// LS Electric XG5000 project: 16-45-1
// PLC NewPLC
// module base 0 slot 0: 입출력 모듈:XBC-DR14E (DC 24V 입력 8점, 릴레이 출력 6점)

PROGRAM NewProgram (task: 스캔 프로그램)

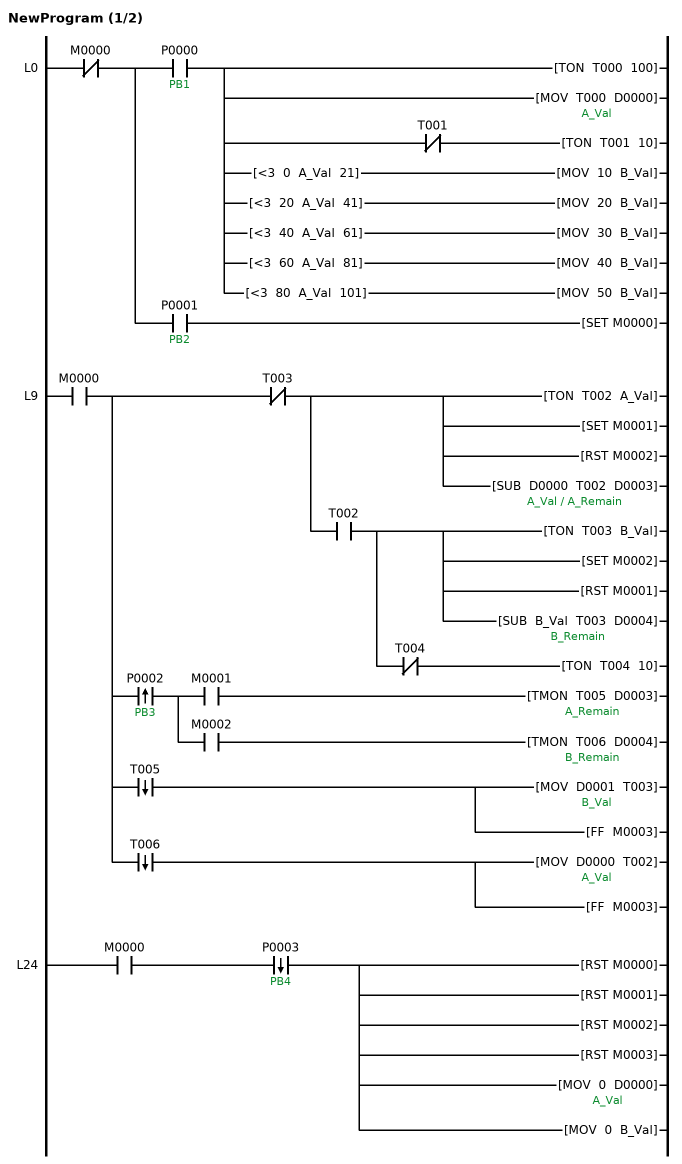
; L0
LOAD NOT  M0000
MPUSH
AND       P0000	// PB1
TON       T000 100
MOV       T000 D0000	// A_Val
MPUSH
AND NOT   T001
TON       T001 10
MLOAD
AND<3     0 A_Val 21
MOV       10 B_Val
MLOAD
AND<3     20 A_Val 41
MOV       20 B_Val
MLOAD
AND<3     40 A_Val 61
MOV       30 B_Val
MLOAD
AND<3     60 A_Val 81
MOV       40 B_Val
MPOP
AND<3     80 A_Val 101
MOV       50 B_Val
MPOP
AND       P0001	// PB2
SET       M0000
; L9
LOAD      M0000
MPUSH
AND NOT   T003
TON       T002 A_Val
SET       M0001
RST       M0002
SUB       D0000 T002 D0003	// A_Val / A_Remain
AND       T002
TON       T003 B_Val
SET       M0002
RST       M0001
SUB       B_Val T003 D0004	// B_Remain
AND NOT   T004
TON       T004 10
MLOAD
ANDP      P0002	// PB3
MPUSH
AND       M0001
TMON      T005 D0003	// A_Remain
MPOP
AND       M0002
TMON      T006 D0004	// B_Remain
MLOAD
ANDN      T005
MOV       D0001 T003	// B_Val
FF        M0003
MPOP
ANDN      T006
MOV       D0000 T002	// A_Val
FF        M0003
; L24
LOAD      M0000
ANDN      P0003	// PB4
RST       M0000
RST       M0001
RST       M0002
RST       M0003
MOV       0 D0000	// A_Val
MOV       0 B_Val

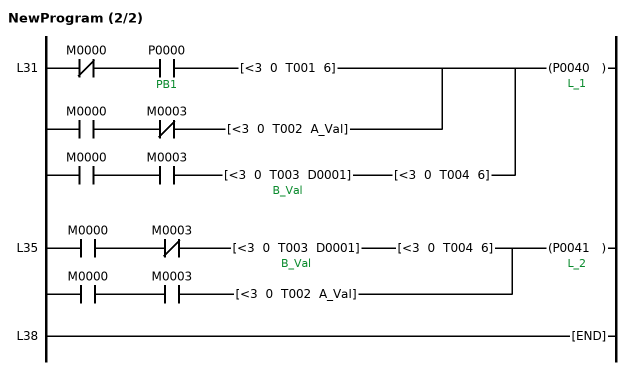
; L31
LOAD NOT  M0000
AND       P0000	// PB1
AND<3     0 T001 6
LOAD      M0000
AND NOT   M0003
AND<3     0 T002 A_Val
OR LOAD
LOAD      M0000
AND       M0003
AND<3     0 T003 D0001	// B_Val
AND<3     0 T004 6
OR LOAD
OUT       P0040	// L_1
; L35
LOAD      M0000
AND NOT   M0003
AND<3     0 T003 D0001	// B_Val
AND<3     0 T004 6
LOAD      M0000
AND       M0003
AND<3     0 T002 A_Val
OR LOAD
OUT       P0041	// L_2
; L38
END